(* IEC 61131-3 sources: Lasal/CPU_5344_V01/Class/cntrTime, 1 file *)

(* ---- cntrTime.st ---- *)
(*!
<Class
	Name               = "cntrTime"
	Revision           = "0.0"
	RealtimeTask       = "false"
	CyclicTask         = "false"
	BackgroundTask     = "true"
	DefBackground      = "10 ms"
	Sigmatek           = "false"
	OSInterface        = "false"
	HighPriority       = "false"
	Automatic          = "false"
	UpdateMode         = "Prescan"
	SharedCommandTable = "true"
	Objectsize         = "(284,120)">
	<Channels>
		<Server Name="ClassSvr" Visualized="false" Initialize="false" WriteProtected="true" Retentive="false"/>
		<Server Name="resetSoftCounter" Visualized="true" Initialize="false" WriteProtected="false" Retentive="false"/>
		<Server Name="softCntrHr" Visualized="true" Initialize="false" WriteProtected="true" Retentive="false"/>
		<Server Name="softCounter" Visualized="false" Initialize="false" WriteProtected="false" Retentive="SRam"/>
		<Server Name="totalCounter" Visualized="false" Initialize="false" WriteProtected="false" Retentive="SRam"/>
		<Server Name="totalCounterHr" Visualized="true" Initialize="false" WriteProtected="true" Retentive="false"/>
		<Client Name="active" Required="false" Internal="false"/>
	</Channels>
</Class>
*)
cntrTime : CLASS
  //Servers:
	ClassSvr 	: SvrChCmd_DINT;
	softCounter 	: SvrCh_DINT;
	totalCounter 	: SvrCh_DINT;
	resetSoftCounter 	: SvrCh_DINT;
	softCntrHr 	: SvrCh_DINT;
	totalCounterHr 	: SvrCh_DINT;
  //Clients:
	active 	: CltCh_DINT;
  //Variables:
		timeActive 	: UDINT;
		timeWritten 	: UDINT;
		tmpCounter 	: DINT;
  //Functions:

	FUNCTION VIRTUAL GLOBAL Init;

	FUNCTION VIRTUAL GLOBAL Background
		VAR_INPUT
			EAX 	: UDINT;
		END_VAR
		VAR_OUTPUT
			state (EAX) 	: UDINT := READY;
		END_VAR;

	FUNCTION storeIt;

	FUNCTION VIRTUAL GLOBAL resetSoftCounter::Write
		VAR_INPUT
			input (EAX) 	: DINT;
		END_VAR
		VAR_OUTPUT
			result (EAX) 	: DINT;
		END_VAR;
  //Tables:
	FUNCTION @STD
		VAR_OUTPUT
			ret_code	: CONFSTATES;
		END_VAR;
	FUNCTION GLOBAL TAB @CT_;
END_CLASS;

// JdK 21-11-2019: class to count time something like a motor is on, they are stored in ram servers, don't write them to often

FUNCTION VIRTUAL GLOBAL cntrTime::Init

  tmpCounter:= totalCounter;

END_FUNCTION

FUNCTION VIRTUAL GLOBAL cntrTime::Background
	VAR_INPUT
		EAX 	: UDINT;
	END_VAR
	VAR_OUTPUT
		state (EAX) 	: UDINT;(* := READY *)
	END_VAR

  active:= active.Read();
  IF active= 0 THEN
    timeActive:= ops.tAbsolute;
  ELSIF ops.tAbsolute-timeActive > 100 THEN //store every 0.1 second
    softCounter+= 1;
    totalCounter+= 1;
    timeActive+= 100;

    IF totalCounter-tmpCounter > 1200 THEN //store every 2 minutes
      storeIt();
    END_IF;

  END_IF;

  IF totalCounter = tmpCounter THEN
    timeWritten:= ops.tAbsolute;
  ELSIF ops.tAbsolute-timeWritten > 300000 THEN //after 5 minutes
    storeIt();
  END_IF;

  softCntrHr:=softCounter/3600; //in 1/10 hr
  totalCounterHr:=totalCounter/3600;

END_FUNCTION

FUNCTION cntrTime::storeIt

  tmpCounter:=totalCounter;
  softCounter-= 1; //we can only store a new value
  totalCounter-= 1;
  softCounter.Write(input:=softCounter+1); //write action to store value
  totalCounter.Write(input:=totalCounter+1);

END_FUNCTION

FUNCTION VIRTUAL GLOBAL cntrTime::resetSoftCounter::Write
	VAR_INPUT
		input (EAX) 	: DINT;
	END_VAR
	VAR_OUTPUT
		result (EAX) 	: DINT;
	END_VAR

	resetSoftCounter := input;
  softCounter.Write(input:=0);
	result := resetSoftCounter;

END_FUNCTION
